{attribute 'TcGenerated'}
{attribute 'no-analysis'}
{attribute 'linkalways'}
// This function has been automatically generated from the project information.
VAR_GLOBAL CONSTANT
	{attribute 'const_non_replaced'}
	stLibVersion_TwinCAT_Open_Framework_Automation_Engine : ST_LibVersion := (iMajor := 1, iMinor := 0, iBuild := 2, iRevision := 0, nFlags := 0, sVersion := '1.0.2.0');
END_VAR

(* stored: Version 1.1.0.1
   GVL Global_Version: Id {48e94b1f-52d4-460e-8b68-1f6cbbb46c37} *)
